FUNCTION INTERNAL _Cleanup
VAR
	i					: UDINT;
	_iSignal			: I_SignalNode;
END_VAR

// Loop through stEntry to update signal ids
FOR i := 1 TO Param.nChannelSize DO
	IF _Channel.stEntry[i].iSignal <> 0 AND_THEN _Channel.stEntry[i].iSignal <> _iSignal THEN
			_iSignal := _Channel.stEntry[i].iSignal;
			_iSignal.id := i;
	END_IF
END_FOR

END_FUNCTION

(* stored: Version 1.1.0.1
   POU _Cleanup: Id {2a20a463-c817-4833-9c12-1d87fdc2ac90}, SpecialFunc None *)
